// TIA Portal V17 export
// export: Created 2025-06-17T13:10:25.6698013Z, ExportSetting WithDefaults, DisplayName Totally Integrated Automation Portal, DisplayVersion V17, DisplayName TIA Portal Openness, DisplayVersion V17, DisplayName TIA Portal Teamcenter Gateway, DisplayVersion V17, DisplayName TIA Portal Version Control Interface, DisplayVersion V17, DisplayName TIA Portal Test Suite Advanced, DisplayVersion V17, DisplayName STEP 7 Professional, DisplayVersion V17, DisplayName STEP 7 Safety, DisplayVersion V17, DisplayName WinCC Advanced / Unified PC, DisplayVersion V17
VAR_GLOBAL   // PLC tag table "Default tag table"
   "high sensor" AT %I0.0 : Bool;
   "low sensor" AT %I0.1 : Bool;
   "pallet sensor" AT %I0.2 : Bool;
   "loaded sensor" AT %I0.3 : Bool;
   "at the left entry" AT %I0.4 : Bool;
   "at the left exit" AT %I0.5 : Bool;
   "at right entry" AT %I0.6 : Bool;
   "at right exit" AT %I0.7 : Bool;
   start AT %I1.0 : Bool;
   reset AT %I1.1 : Bool;
   stop AT %I1.2 : Bool;
   "Emergency stop" AT %I1.3 : Bool;
   auto AT %I1.4 : Bool;
   "factory runnning" AT %I1.5 : Bool;
   "conveyor enter" AT %Q0.0 : Bool;
   load AT %Q0.1 : Bool;
   unload AT %Q0.2 : Bool;
   "transfer left" AT %Q0.3 : Bool;
   "transfer right" AT %Q0.4 : Bool;
   "conveyor left" AT %Q0.5 : Bool;
   "conveyor right" AT %Q0.6 : Bool;
   "start light" AT %Q0.7 : Bool;
   "Reset light" AT %Q1.0 : Bool;
   "stop light" AT %Q1.1 : Bool;
   "counter" AT %QW30 : Int;
END_VAR
